// TIA Portal V17 export
// export: Created 2026-04-13T11:12:41.7222797Z, ExportSetting WithDefaults, DisplayName Totally Integrated Automation Portal, DisplayVersion V17 Update 4, DisplayName TIA Portal Openness, DisplayVersion V17 Update 4, DisplayName TIA Portal Version Control Interface, DisplayVersion V17, DisplayName SINAMICS Startdrive Advanced, DisplayVersion V17, DisplayName SINAMICS Startdrive G130, G150, S120, S150, SINAMICS MV, S210, DisplayVersion V17, DisplayName SINAMICS Startdrive G110M, G120, G120C, G120D, G120P, G115D, DisplayVersion V17, DisplayName STEP 7 Professional, DisplayVersion V17 Update 4, DisplayName STEP 7 Safety, DisplayVersion V17, DisplayName WinCC Professional, DisplayVersion V17 Update 4
FUNCTION_BLOCK "A7-通信心跳块"   // FB14, SCL
{ S7_Optimized_Access := 'TRUE' }
VERSION : 0.1
// stored: AutoNumber true, IsIECCheckEnabled false, IsRetainMemResEnabled false, MemoryReserve 100, SetENOAutomatically false, UDAEnableTagReadback false
   VAR_OUTPUT
      通信失联 : Bool;
   END_VAR
   VAR_IN_OUT
      real_SC输出值 : Real;
      real_FK反馈值 : Real;
      超时时间 : Time := T#120S;
      i : Int;
   END_VAR
   VAR RETAIN
      t1 : TON_TIME;
      t2 { S7_SetPoint := 'True'} : TON_TIME;
   END_VAR
   VAR
      RT1 : R_TRIG;
   END_VAR
   VAR RETAIN
      间隔时间 : Time := T#5S;
      SC输出值 : Int;
      FK反馈值 : Int;
   END_VAR
   VAR_TEMP
      TM_FZ : Int;
   END_VAR
BEGIN
   #TM_FZ := #FK反馈值;

   #SC输出值 := REAL_TO_INT(#real_SC输出值);
   #FK反馈值 := REAL_TO_INT(#real_FK反馈值);

   #t1(IN := (#TM_FZ <> #SC输出值) ,
       PT := #超时时间,
       Q=>#通信失联);


   (* IF #t1.Q THEN
       (* #TM_FZ := 1; *)
       #SC输出值 := #SC输出值 - 1;
   END_IF; *)

   IF #TM_FZ = #SC输出值 THEN

       IF #SC输出值 MOD 2 = 0 THEN

           #SC输出值 := #SC输出值 + 1;
       ELSE

           #SC输出值 := #SC输出值 - 1;
       END_IF;

   END_IF;
END_FUNCTION_BLOCK
